TYPE ST_RxUdpRemote :
STRUCT
	comau : ST_ComauControl;
END_STRUCT
END_TYPE

(* stored: Version 1.1.0.1, ProductVersion 3.1.4022.7
   DUT ST_RxUdpRemote: Id {73287563-87c0-4e8c-8c64-be7e0b2fa243} *)
